PROGRAM FullProcess
VAR
END_VAR
// written 7.08.2023 by Daniel Kelly

// This program is the full version of the process. It includes longer feeding 
// and residence times
// RValveOff turns off the solenoids on the righthandside incase they were already on
// OpenValve opens the top valve
// Step Vacuum removes the excess air from inside the pipe via the vacuum
//waitTemp waits until the temperature is at least 350 degrees celsius
// BiomassFeed operates the second feeding motor
// Init_Feed operates the main feeding motor
// wait600 waits until temperature is 600
// GasFanON turns on the gas fan
// ShortFeed turns on the main feeding motor 1
// ExitMotor turns on the removal motor and opens the top valve
// Valve2Open opens the bottom valve
// Valve2Close closes the bottom valve
// SolenoidsOff turns off the solenoids incase they were on
// AirRemoval removes the air from the pipe
// turnoff1 etc. turns off the devices such as the valves and feeding motor 2

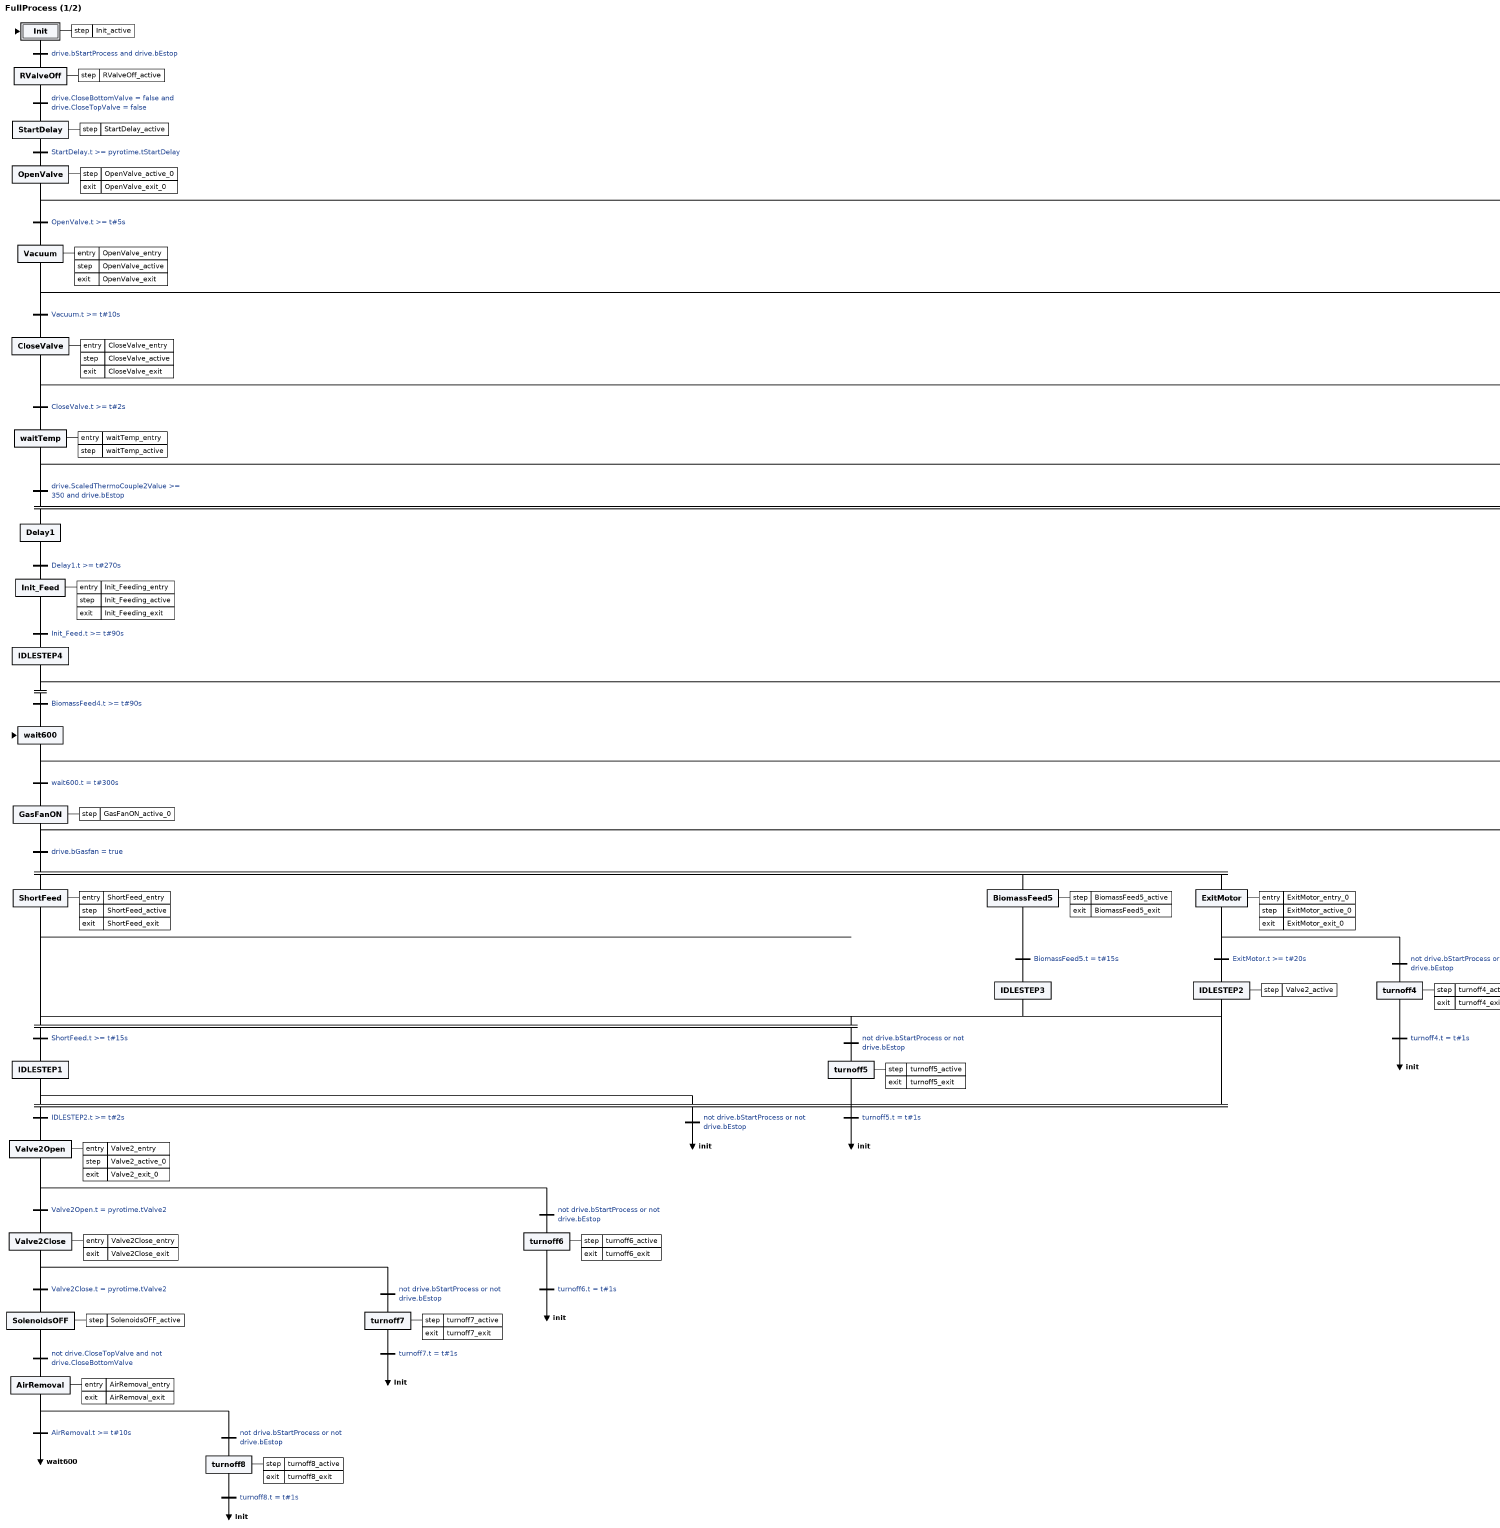
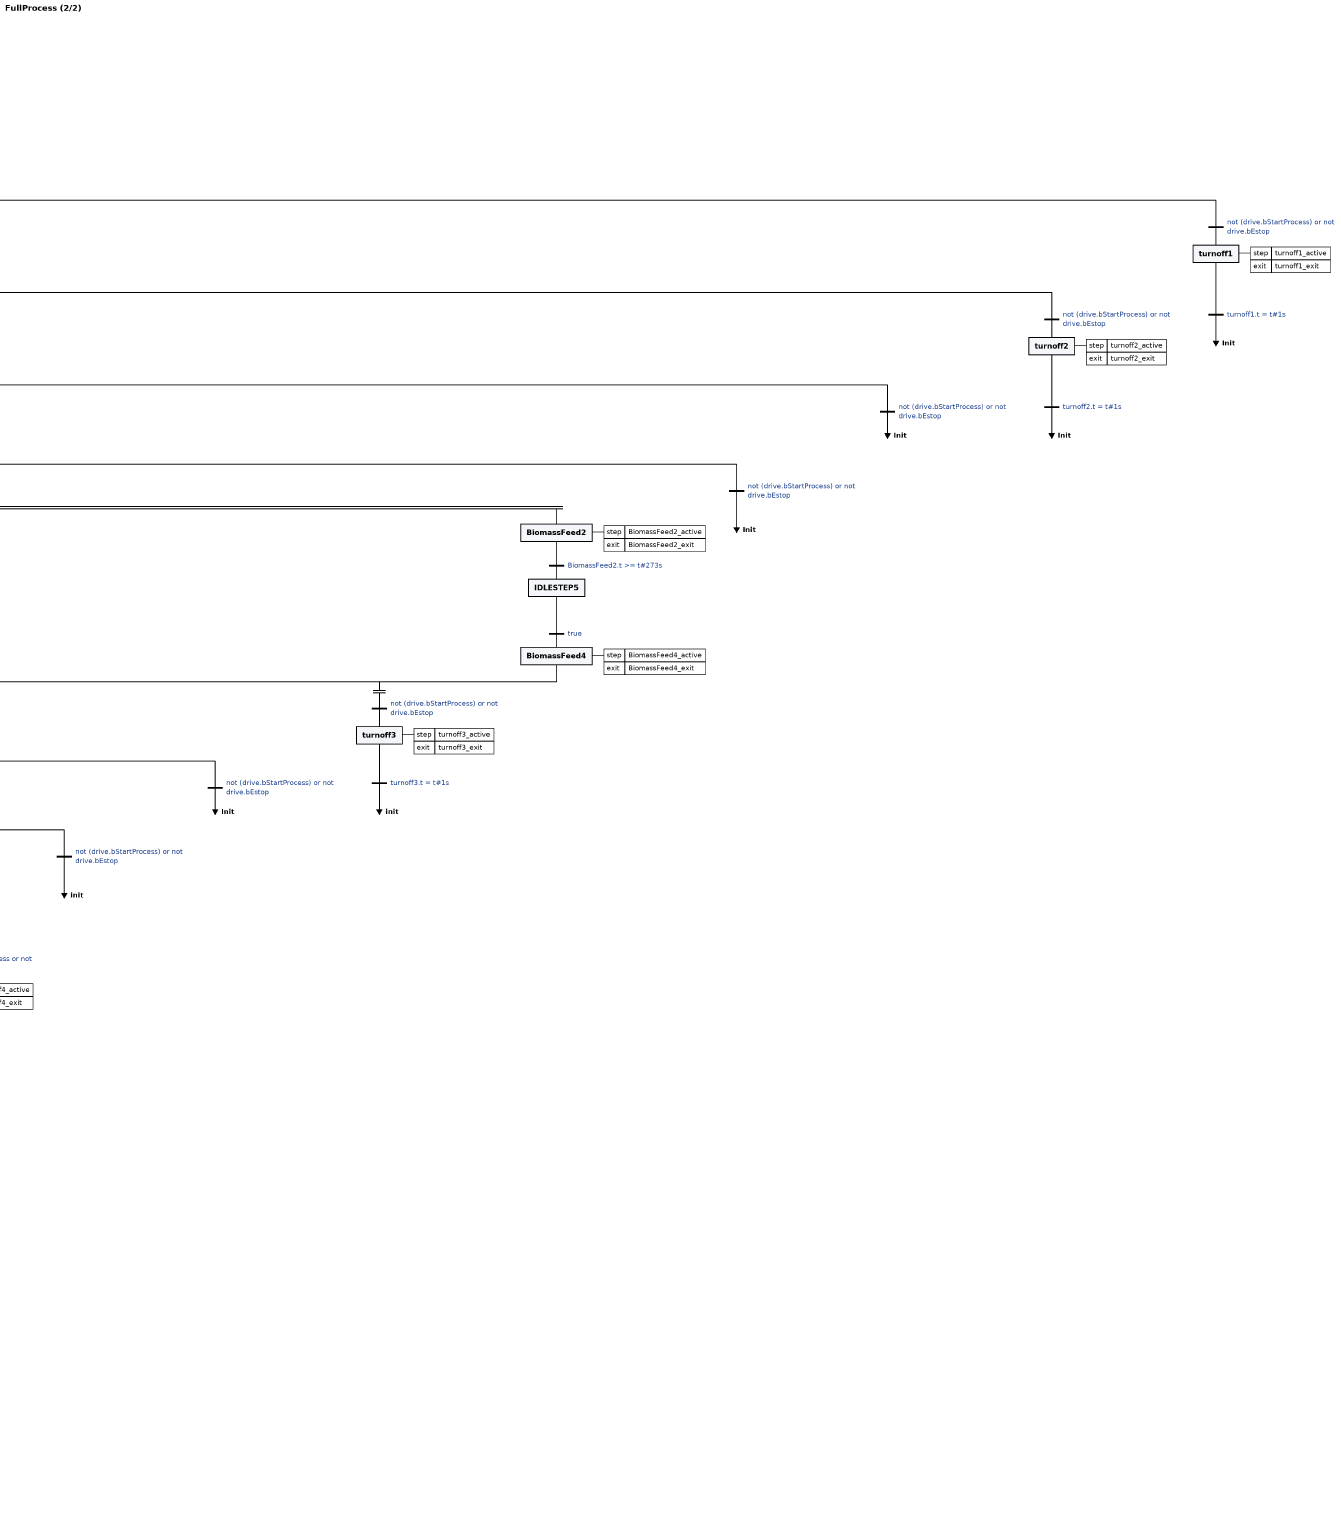
INITIAL_STEP Init:
    Init_active(N);  // step action
END_STEP
TRANSITION FROM Init TO RValveOff
    := drive.bStartProcess and drive.bEstop;
END_TRANSITION
STEP RValveOff:
    RValveOff_active(N);  // step action
END_STEP
TRANSITION FROM RValveOff TO StartDelay
    := drive.CloseBottomValve = false and drive.CloseTopValve = false;
END_TRANSITION
STEP StartDelay:
    StartDelay_active(N);  // step action
END_STEP
TRANSITION FROM StartDelay TO OpenValve
    := StartDelay.t >= pyrotime.tStartDelay;
END_TRANSITION
STEP OpenValve:
    OpenValve_active_0(N);  // step action
    OpenValve_exit_0(P0);  // exit action
END_STEP
TRANSITION FROM OpenValve TO Vacuum
    := OpenValve.t >= t#5s;
END_TRANSITION
TRANSITION FROM OpenValve TO turnoff1
    := not (drive.bStartProcess) or not drive.bEstop;
END_TRANSITION
STEP turnoff1:
    turnoff1_active(N);  // step action
    turnoff1_exit(P0);  // exit action
END_STEP
TRANSITION FROM turnoff1 TO Init
    := turnoff1.t = t#1s;
END_TRANSITION
STEP Vacuum:
    OpenValve_entry(P1);  // entry action
    OpenValve_active(N);  // step action
    OpenValve_exit(P0);  // exit action
END_STEP
TRANSITION FROM Vacuum TO CloseValve
    := Vacuum.t >= t#10s;
END_TRANSITION
TRANSITION FROM Vacuum TO turnoff2
    := not (drive.bStartProcess) or not drive.bEstop;
END_TRANSITION
STEP turnoff2:
    turnoff2_active(N);  // step action
    turnoff2_exit(P0);  // exit action
END_STEP
TRANSITION FROM turnoff2 TO Init
    := turnoff2.t = t#1s;
END_TRANSITION
STEP CloseValve:
    CloseValve_entry(P1);  // entry action
    CloseValve_active(N);  // step action
    CloseValve_exit(P0);  // exit action
END_STEP
TRANSITION FROM CloseValve TO waitTemp
    := CloseValve.t >= t#2s;
END_TRANSITION
TRANSITION FROM CloseValve TO Init
    := not (drive.bStartProcess) or not drive.bEstop;
END_TRANSITION
STEP waitTemp:
    waitTemp_entry(P1);  // entry action
    waitTemp_active(N);  // step action
END_STEP
TRANSITION FROM waitTemp TO (Delay1, BiomassFeed2)
    := drive.ScaledThermoCouple2Value >= 350 and drive.bEstop;
END_TRANSITION
TRANSITION FROM waitTemp TO Init
    := not (drive.bStartProcess) or not drive.bEstop;
END_TRANSITION
STEP Delay1:
END_STEP
TRANSITION FROM Delay1 TO Init_Feed
    := Delay1.t >= t#270s;
END_TRANSITION
STEP Init_Feed:
    Init_Feeding_entry(P1);  // entry action
    Init_Feeding_active(N);  // step action
    Init_Feeding_exit(P0);  // exit action
END_STEP
TRANSITION FROM Init_Feed TO IDLESTEP4
    := Init_Feed.t >= t#90s;
END_TRANSITION
STEP IDLESTEP4:
END_STEP
STEP BiomassFeed2:
    BiomassFeed2_active(N);  // step action
    BiomassFeed2_exit(P0);  // exit action
END_STEP
TRANSITION FROM BiomassFeed2 TO IDLESTEP5
    := BiomassFeed2.t >= t#273s;
END_TRANSITION
STEP IDLESTEP5:
END_STEP
TRANSITION FROM IDLESTEP5 TO BiomassFeed4
    := true;
END_TRANSITION
STEP BiomassFeed4:
    BiomassFeed4_active(N);  // step action
    BiomassFeed4_exit(P0);  // exit action
END_STEP
TRANSITION FROM (IDLESTEP4, BiomassFeed4) TO wait600
    := BiomassFeed4.t >= t#90s;
END_TRANSITION
TRANSITION FROM (IDLESTEP4, BiomassFeed4) TO turnoff3
    := not (drive.bStartProcess) or not drive.bEstop;
END_TRANSITION
STEP turnoff3:
    turnoff3_active(N);  // step action
    turnoff3_exit(P0);  // exit action
END_STEP
TRANSITION FROM turnoff3 TO init
    := turnoff3.t = t#1s;
END_TRANSITION
STEP wait600:
END_STEP
TRANSITION FROM wait600 TO GasFanON
    := wait600.t = t#300s;
END_TRANSITION
STEP GasFanON:
    GasFanON_active_0(N);  // step action
END_STEP
TRANSITION FROM GasFanON TO (ShortFeed, BiomassFeed5, ExitMotor)
    := drive.bGasfan = true;
END_TRANSITION
TRANSITION FROM GasFanON TO init
    := not (drive.bStartProcess) or not drive.bEstop;
END_TRANSITION
TRANSITION FROM wait600 TO Init
    := not (drive.bStartProcess) or not drive.bEstop;
END_TRANSITION
STEP ShortFeed:
    ShortFeed_entry(P1);  // entry action
    ShortFeed_active(N);  // step action
    ShortFeed_exit(P0);  // exit action
END_STEP
STEP BiomassFeed5:
    BiomassFeed5_active(N);  // step action
    BiomassFeed5_exit(P0);  // exit action
END_STEP
TRANSITION FROM BiomassFeed5 TO IDLESTEP3
    := BiomassFeed5.t = t#15s;
END_TRANSITION
STEP IDLESTEP3:
END_STEP
TRANSITION FROM (ShortFeed, IDLESTEP3) TO IDLESTEP1
    := ShortFeed.t >= t#15s;
END_TRANSITION
TRANSITION FROM (ShortFeed, IDLESTEP3) TO turnoff5
    := not drive.bStartProcess or not drive.bEstop;
END_TRANSITION
STEP turnoff5:
    turnoff5_active(N);  // step action
    turnoff5_exit(P0);  // exit action
END_STEP
TRANSITION FROM turnoff5 TO init
    := turnoff5.t = t#1s;
END_TRANSITION
STEP IDLESTEP1:
END_STEP
STEP ExitMotor:
    ExitMotor_entry_0(P1);  // entry action
    ExitMotor_active_0(N);  // step action
    ExitMotor_exit_0(P0);  // exit action
END_STEP
TRANSITION FROM ExitMotor TO IDLESTEP2
    := ExitMotor.t >= t#20s;
END_TRANSITION
TRANSITION FROM ExitMotor TO turnoff4
    := not drive.bStartProcess or not drive.bEstop;
END_TRANSITION
STEP turnoff4:
    turnoff4_active(N);  // step action
    turnoff4_exit(P0);  // exit action
END_STEP
TRANSITION FROM turnoff4 TO init
    := turnoff4.t = t#1s;
END_TRANSITION
STEP IDLESTEP2:
    Valve2_active(N);  // step action
END_STEP
TRANSITION FROM (IDLESTEP1, IDLESTEP2) TO Valve2Open
    := IDLESTEP2.t >= t#2s;
END_TRANSITION
TRANSITION FROM (IDLESTEP1, IDLESTEP2) TO init
    := not drive.bStartProcess or not drive.bEstop;
END_TRANSITION
STEP Valve2Open:
    Valve2_entry(P1);  // entry action
    Valve2_active_0(N);  // step action
    Valve2_exit_0(P0);  // exit action
END_STEP
TRANSITION FROM Valve2Open TO Valve2Close
    := Valve2Open.t = pyrotime.tValve2;
END_TRANSITION
TRANSITION FROM Valve2Open TO turnoff6
    := not drive.bStartProcess or not drive.bEstop;
END_TRANSITION
STEP turnoff6:
    turnoff6_active(N);  // step action
    turnoff6_exit(P0);  // exit action
END_STEP
TRANSITION FROM turnoff6 TO init
    := turnoff6.t = t#1s;
END_TRANSITION
STEP Valve2Close:
    Valve2Close_entry(P1);  // entry action
    Valve2Close_exit(P0);  // exit action
END_STEP
TRANSITION FROM Valve2Close TO SolenoidsOFF
    := Valve2Close.t = pyrotime.tValve2;
END_TRANSITION
TRANSITION FROM Valve2Close TO turnoff7
    := not drive.bStartProcess or not drive.bEstop;
END_TRANSITION
STEP turnoff7:
    turnoff7_active(N);  // step action
    turnoff7_exit(P0);  // exit action
END_STEP
TRANSITION FROM turnoff7 TO Init
    := turnoff7.t = t#1s;
END_TRANSITION
STEP SolenoidsOFF:
    SolenoidsOFF_active(N);  // step action
END_STEP
TRANSITION FROM SolenoidsOFF TO AirRemoval
    := not drive.CloseTopValve and not drive.CloseBottomValve;
END_TRANSITION
STEP AirRemoval:
    AirRemoval_entry(P1);  // entry action
    AirRemoval_exit(P0);  // exit action
END_STEP
TRANSITION FROM AirRemoval TO wait600
    := AirRemoval.t >= t#10s;
END_TRANSITION
TRANSITION FROM AirRemoval TO turnoff8
    := not drive.bStartProcess or not drive.bEstop;
END_TRANSITION
STEP turnoff8:
    turnoff8_active(N);  // step action
    turnoff8_exit(P0);  // exit action
END_STEP
TRANSITION FROM turnoff8 TO Init
    := turnoff8.t = t#1s;
END_TRANSITION

ACTION AirRemoval_entry:
drive.bVacuum := TRUE;
END_ACTION

ACTION AirRemoval_exit:
drive.bVacuum := FALSE;
END_ACTION

ACTION BiomassFeed_active:
drive.bFeedMotor2 := true;
END_ACTION

ACTION BiomassFeed_exit:
drive.bFeedMotor2 := false;
END_ACTION

ACTION BiomassFeed2_active:
drive.bFeedMotor2 := TRUE;
END_ACTION

ACTION BiomassFeed2_exit:
drive.bFeedMotor2 := FALSE;
END_ACTION

ACTION BiomassFeed4_active:
drive.bFeedMotor2 := TRUE;
END_ACTION

ACTION BiomassFeed4_exit:
drive.bFeedMotor2 := false;
END_ACTION

ACTION BiomassFeed5_active:
drive.bFeedMotor2 := true;
END_ACTION

ACTION BiomassFeed5_exit:
drive.bFeedMotor2 := false;
END_ACTION

ACTION CloseValve_active:
drive.CloseTopValve := TRUE;
drive.CloseBottomValve := FALSE;
END_ACTION

ACTION CloseValve_entry:
//drive.RightSolenoid := TRUE;
END_ACTION

ACTION CloseValve_exit:
drive.CloseTopValve := FALSE;
END_ACTION

ACTION ExitMotor_active_0:
drive.bRemovalMotor := TRUE;
drive.bM2active := TRUE; // lamp variable



drive.OpenTopValve := TRUE; // opens valve
drive.CloseTopValve := FALSE;
END_ACTION

ACTION ExitMotor_entry_0:

END_ACTION

ACTION ExitMotor_exit_0:
 
drive.CloseTopValve := TRUE; //closes valve
drive.OpenTopValve := FALSE;

drive.bM2active := FALSE; // lamp variable ; turns lamp off
drive.bRemovalMotor := FALSE; // turns the removal motor off
END_ACTION

ACTION ExitMotor1_active:
drive.bRemovalMotor := TRUE;
END_ACTION

ACTION GasFanOFF_active:
drive.bGasfan := false;
END_ACTION

ACTION GasFanOFF_active_0:
drive.bGasfan := false;
END_ACTION

ACTION GasFanOn_active:
drive.bGasfan := TRUE;
END_ACTION

ACTION GasFanON_active_0:
drive.bGasfan := TRUE;
END_ACTION

ACTION Init_active:
//drive.ATV_RPDO_Output1_Control_Word := 0;
//drive.bRemovalMotor := FALSE; 
//drive.bProcessActive := FALSE;
//drive.LeftSolenoid := FALSE;
//drive.LeftSolenoid2 := FALSE; 
//drive.RightSolenoid := TRUE;
//drive.RightSolenoid2 := TRUE;
 
drive.ifeedmotor1count := 0;
END_ACTION

ACTION Init_Feeding_active:
IF drive.ATV_TPDO_Input1_Status_Word = ATV_Status.rdy2SwitchON THEN 
	drive.ATV_RPDO_Output1_Control_Word := 7; //SwitchedON
END_IF

IF drive.ATV_TPDO_Input1_Status_Word = ATV_Status.SwitchedON THEN 
	drive.ATV_RPDO_Output1_Control_Word := 15; //OP_Enabled
	drive.bM1active := TRUE; // lamp goes on
	drive.bM1status := TRUE;  // status variable
END_IF
END_ACTION

ACTION Init_Feeding_entry:
drive.ATV_RPDO_Output1_Control_Word := 6; //rdy2SwitchON
drive.ATV_RPDO_Output2_Target_Velocity := 1000;
END_ACTION

ACTION Init_Feeding_exit:


IF drive.bM1status = TRUE THEN 
	drive.ifeedmotor1count := drive.ifeedmotor1count + 1;
END_IF

drive.ATV_RPDO_Output1_Control_Word := 7; //switchedON, ready mode
drive.bM1active := FALSE;  // lamp off
drive.bM1status := FALSE;  // status variable for feeding motor 1
END_ACTION

ACTION OpenValve_active:

END_ACTION

ACTION OpenValve_active_0:
drive.OpenTopValve := TRUE;
drive.CloseTopValve := FALSE;
END_ACTION

ACTION OpenValve_entry:

drive.bVacuum := TRUE;
END_ACTION

ACTION OpenValve_exit:
drive.bVacuum := FALSE;
END_ACTION

ACTION OpenValve_exit_0:
drive.OpenTopValve := false;
END_ACTION

ACTION ProcessActive_active:
IF drive.bStartProcess THEN 
	drive.bProcessActive := TRUE;
ELSE 
	drive.bProcessActive := FALSE; 
END_IF
END_ACTION

ACTION RValveOff_active:
drive.CloseTopValve := FALSE;
drive.CloseBottomValve := FALSE;
END_ACTION

ACTION ShortFeed_active:
IF drive.ATV_TPDO_Input1_Status_Word = ATV_Status.rdy2SwitchON THEN 
	drive.ATV_RPDO_Output1_Control_Word := 7;
END_IF

IF drive.ATV_TPDO_Input1_Status_Word = ATV_Status.SwitchedON THEN
			drive.bM1run := TRUE; //counter variable
			drive.bM1active := TRUE;
			drive.ATV_RPDO_Output1_Control_Word := 15;
END_IF
END_ACTION

ACTION ShortFeed_entry:
drive.ATV_RPDO_Output2_Target_Velocity := 1000;
drive.ATV_RPDO_Output1_Control_Word := 6;
END_ACTION

ACTION ShortFeed_exit:


drive.bM1run := FALSE;
drive.bM1active := FALSE; 
drive.ATV_RPDO_Output1_Control_Word := 7;
END_ACTION

ACTION SolenoidsOFF_active:
drive.CloseTopValve := FALSE;
drive.CloseBottomValve := FALSE;
END_ACTION

ACTION StartDelay_active:
IF drive.bStartProcess THEN 
	drive.bProcessActive := TRUE;
ELSE 
	drive.bProcessActive := FALSE; 
END_IF
END_ACTION

ACTION turnoff1_active:
drive.CloseTopValve := TRUE;
drive.OpenTopValve := FALSE;
END_ACTION

ACTION turnoff1_exit:
drive.CloseTopValve := FALSE;
END_ACTION

ACTION turnoff2_active:
drive.bVacuum := FALSE;
END_ACTION

ACTION turnoff2_exit:

END_ACTION

ACTION turnoff3_active:
drive.bM1status := FALSE;
drive.bFeedMotor2 := FALSE;
drive.bM1active := FALSE;
END_ACTION

ACTION turnoff3_exit:

END_ACTION

ACTION turnoff4_active:
drive.bRemovalMotor := FALSE;
drive.bM2active := FALSE;

drive.OpenTopValve := FALSE;
drive.CloseTopValve := TRUE;
END_ACTION

ACTION turnoff4_exit:
drive.CloseTopValve := false;
END_ACTION

ACTION turnoff5_active:
drive.bFeedMotor2 := FALSE;


drive.bRemovalMotor := FALSE;
drive.bM2active := FALSE;

drive.OpenTopValve := FALSE;
drive.CloseTopValve := TRUE;
END_ACTION

ACTION turnoff5_exit:

END_ACTION

ACTION turnoff6_active:
drive.CloseBottomValve := TRUE;
drive.OpenBottomValve := FALSE;
END_ACTION

ACTION turnoff6_exit:
drive.CloseBottomValve := FALSE;
END_ACTION

ACTION turnoff7_active:
drive.CloseBottomValve := TRUE;
END_ACTION

ACTION turnoff7_exit:
drive.CloseBottomValve := FALSE;
END_ACTION

ACTION turnoff8_active:
drive.bVacuum := false;
END_ACTION

ACTION turnoff8_exit:

END_ACTION

ACTION Vacuum_entry:

END_ACTION

ACTION Vacuum_exit:
drive.bVacuum := FALSE;
END_ACTION

ACTION Valve2_active:

END_ACTION

ACTION Valve2_active_0:

END_ACTION

ACTION Valve2_entry:
drive.OpenBottomValve := TRUE;
END_ACTION

ACTION Valve2_exit_0:
drive.OpenBottomValve := FALSE;
END_ACTION

ACTION Valve2Close_entry:
drive.CloseBottomValve := TRUE;
END_ACTION

ACTION Valve2Close_exit:
 drive.CloseBottomValve := FALSE;
END_ACTION

ACTION waitTemp_active:

END_ACTION

ACTION waitTemp_entry:

END_ACTION

END_PROGRAM

(* stored: Version 1.1.0.1, ProductVersion 3.1.4024.12
   POU FullProcess: Id {a5bbb2c4-a56b-45fc-8307-6a99f2ed9c34}, SpecialFunc None
   Action AirRemoval_entry: Id {56986495-ea09-45bf-8c82-62a4887e6ffc}
   Action AirRemoval_exit: Id {3bddf684-ae8b-410c-95fd-58b384a4d056}
   Action BiomassFeed_active: Id {db361a60-5c0f-46d8-a1e6-813e6bcaa0a6}
   Action BiomassFeed_exit: Id {626386fe-4ef9-4c7b-abbf-ea540ca57cb1}
   Action BiomassFeed2_active: Id {7203e835-d662-4e3c-9656-6254cd70714e}
   Action BiomassFeed2_exit: Id {11c4385b-2c20-4732-b513-55a8ecff74fc}
   Action BiomassFeed4_active: Id {241fdc92-aa3f-4cb0-a818-5f92c37f23dc}
   Action BiomassFeed4_exit: Id {7cdc1e81-c650-45e3-b75e-c5c0014f026e}
   Action BiomassFeed5_active: Id {954e17ba-3d15-4f52-adb7-cbd083726f2c}
   Action BiomassFeed5_exit: Id {3ca4c3c7-bcd0-4e81-a9e9-032e199f9fe5}
   Action CloseValve_active: Id {21b9c1c8-71d1-43fa-90a0-09bed8b2be5f}
   Action CloseValve_entry: Id {d65b07a7-c4ae-4873-bd26-ab625000c614}
   Action CloseValve_exit: Id {35a86761-32d5-4569-b629-57df12d6b2da}
   Action ExitMotor_active_0: Id {a4a2b3ca-8e28-4812-862b-9dc6ac0dc1f2}
   Action ExitMotor_entry_0: Id {cf59d1d3-efaa-474b-96c4-01c54da350b1}
   Action ExitMotor_exit_0: Id {4dc62c02-01ca-42d7-98d2-88727f669a7d}
   Action ExitMotor1_active: Id {2160f5eb-ad5f-462a-91c7-8d7eab1527e3}
   Action GasFanOFF_active: Id {dd69af5b-ac20-46ed-ba6b-5be8c9db439b}
   Action GasFanOFF_active_0: Id {54c29cef-9fb9-4d35-9e11-31a42ecffec8}
   Action GasFanOn_active: Id {15c7edf4-89f1-46be-88b2-7870d5ce911a}
   Action GasFanON_active_0: Id {0629d2b9-1b1a-447d-9eda-9b7714f9fd40}
   Action Init_active: Id {8c94ee1e-8c91-4a51-8a83-9d2db698acce}
   Action Init_Feeding_active: Id {fc68ce2d-2718-4a29-a112-65934edc72f2}
   Action Init_Feeding_entry: Id {a7b0eb95-0468-4776-95b7-13c92614e732}
   Action Init_Feeding_exit: Id {85b71a06-c6e3-4261-8b22-448ec9b42f20}
   Action OpenValve_active: Id {a65fb058-b11e-45bd-b454-5c9071c2383e}
   Action OpenValve_active_0: Id {8a0fc9bd-0e9f-43ed-a1d4-54142ea11d21}
   Action OpenValve_entry: Id {7c507d22-66c8-4481-9d56-272620cdb8dd}
   Action OpenValve_exit: Id {f55b26a7-1bad-479e-8466-6917b6e75f5d}
   Action OpenValve_exit_0: Id {57f463aa-3e6c-481b-990e-7119a94440c6}
   Action ProcessActive_active: Id {fcefc1f5-bf85-40f8-b37c-8da98fab6d07}
   Action RValveOff_active: Id {b3f0e466-72fd-4623-a213-0e61618fd4e8}
   Action ShortFeed_active: Id {9d3402e1-0e98-416c-88f1-1c7d0f05f573}
   Action ShortFeed_entry: Id {fd7bcbf3-0919-4cb5-ab51-5ebcdfc7db8e}
   Action ShortFeed_exit: Id {f95b5c24-2d6c-4135-bc68-6ff0b84698db}
   Action SolenoidsOFF_active: Id {979c0249-b5de-4745-a345-880264ea4023}
   Action StartDelay_active: Id {d4a64755-9a8b-400a-bd33-d9f968cb1644}
   Action turnoff1_active: Id {d5df9373-aaea-4a16-9bf0-ed6c62294bd5}
   Action turnoff1_exit: Id {1d910c70-5e3e-447f-ac23-52abadfc30da}
   Action turnoff2_active: Id {0511628f-c949-4197-916d-4d6118ac1dbe}
   Action turnoff2_exit: Id {9642a8fa-c30f-4dcf-bb5f-b09fc0b5e75f}
   Action turnoff3_active: Id {88cc89c3-d19d-44e5-916e-74f2cb97e38e}
   Action turnoff3_exit: Id {e45b3f8d-d110-41cf-8fbe-21d97ee98bc5}
   Action turnoff4_active: Id {e9502fac-6745-425b-ab29-43745e0f400d}
   Action turnoff4_exit: Id {3e2e97be-643b-462e-8dff-3be2e55c13c6}
   Action turnoff5_active: Id {9b04acec-08c0-4194-9539-4bae896d0436}
   Action turnoff5_exit: Id {b565c757-fb4c-4b47-a8c6-6f9f01c2f454}
   Action turnoff6_active: Id {fca560d3-269b-40fb-88d3-a49431481f56}
   Action turnoff6_exit: Id {4cc7a309-2e2f-46ba-a03f-ebd3c3e2ab7c}
   Action turnoff7_active: Id {87d05ac3-54ca-4152-a8b5-d0ca8dc9ad2a}
   Action turnoff7_exit: Id {ba4fbd24-0eec-4b6e-9abd-19c871e8ca7c}
   Action turnoff8_active: Id {e09ce29b-ca82-486e-ab0a-02864e4d9e22}
   Action turnoff8_exit: Id {eae5f9c4-f9e5-46eb-aed0-eda9589b1186}
   Action Vacuum_entry: Id {eada3070-4c9b-4319-8fb2-8bba7df5dfba}
   Action Vacuum_exit: Id {0d5fb7b8-2796-4ab2-8602-aa482adad1b0}
   Action Valve2_active: Id {351cfb2b-e636-4bfb-b930-6532f2bd12a2}
   Action Valve2_active_0: Id {3efcc2cd-e7dd-4e8c-bcbe-03a3b4ea440b}
   Action Valve2_entry: Id {7f970c41-d38d-42eb-8584-009e6235ce83}
   Action Valve2_exit_0: Id {b1cc5001-2875-405b-bb2d-e3d28f67c249}
   Action Valve2Close_entry: Id {cc200eae-3ef3-4e12-89d6-9b3829e74327}
   Action Valve2Close_exit: Id {8ce57674-9c42-4bde-b272-5ad093e9fdcc}
   Action waitTemp_active: Id {500eeb57-b5e8-4213-ad94-45d3791a47fc}
   Action waitTemp_entry: Id {ab2e422d-4cf2-497c-85f2-9a726cf7f851} *)
